FUNCTION_BLOCK OPC_UA_WRITE (* Read value from OPC UA server *)
  (* Standard: OPC UA; Function: Reader *)
  (* Version 1.0, 2015-11-08, Slavomir Kozar, Certicon *)
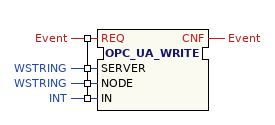
  EVENT_INPUT
    REQ WITH SERVER, NODE, IN; (* Normal Execution Request *)
  END_EVENT
  EVENT_OUTPUT
    CNF; (* Execution Confirmation *)
  END_EVENT
  VAR_INPUT
    SERVER : WSTRING; (* OPC UA server address:port *)
    NODE : WSTRING; (* UPC UA Node ID *)
    IN : INT; (* Data to Write *)
  END_VAR
END_FUNCTION_BLOCK
